INTERFACE I_Serializable EXTENDS __SYSTEM.IQueryInterface

METHOD SerializeWith
VAR_INPUT
	Serializer : I_Serializer;
END_VAR
END_METHOD

END_INTERFACE

(* stored: Version 1.1.0.1, ProductVersion 3.1.4024.12
   Itf I_Serializable: Id {6648b24b-ee2e-4f78-925a-94cc56f9908d}
   Method SerializeWith: Id {2fc6facd-f838-41f6-a46b-87e76fdc57e9} *)
